# EPICS alarm handler configuration: apps/caenScalerApp/alh/watchdogs_nomoller.alhConfig
GROUP    NULL                         HallC_Ops
$GUIDANCE
This alarm panel is intended to alert the operator to various problems
with controls, DAQ and other systems.  If there is some hardware or software
that you think could be included in this panel, please contact Steve Wood.
For this alarm panel to work, vmec15 must be up and healthy.  If most
everything is in an invalid or error state, then reboot vmec15.
$END
GROUP    HallC_Ops                    DataMovement
CHANNEL  DataMovement                 HCDOG_diskwatch
$GUIDANCE
The diskwatch GUI that monitors free disk space is either hung or not
running.  This GUI should be running on the DAQ console.  If it is running,
click the Quit button.  To restart the GUI, type the command "diskwatch"
into an xterm window on the DAQ console.  (Should be logged on as "cdaq").
$END
CHANNEL  DataMovement                 HCDOG_happyreaper
$GUIDANCE
The scripts that copy runs from the data disks to the Silo do not appear
to be running.  Steve Wood should be notified.  However, if there more
than, say, five green partitions in diskwatch, the situation is not
urgent, so don't wake him up in the middle of the night.
$END
GROUP    HallC_Ops                    Monitoring
CHANNEL  Monitoring                   HCDOG_ChannelArchiver
$GUIDANCE
The EPICS Channel Archiver that maintains a continuous log of controls
information is not running.  To restart, logon to jeffylab as "cvxwrks"
 and type the following commands:
	cd ~/Archives
	./stop_archiver
	./start_archiver
$END
CHANNEL  Monitoring                   HCDOG_BetaBrite
$GUIDANCE
The LED display that shows beam current and PSS status is not working
properly.  To restart, logon to jeffylab as "cvxwrks".  Do
"ps -aux | grep bcm_pss" and kill any copies of the script that are
running.  Then type "cd ~/BETABRITE/bcm ; ./bcm_pss.pl&".
$END
GROUP    HallC_Ops                    Crates
$GUIDANCE
The status of many of the counting house NIM bins and Camac crates is
monitored by passing a pulser signal through a module in each crate.
The pulser coming from each crate is connect to an input register.  If
the pulser signal stops for a given crate, an alarm will be raised,
indicating a possible power problem with the crate.
$END
CHANNEL  Crates                       HCDOG_bit0
$GUIDANCE
The watchdog signal from the top NIM bit in rack CH03B05 is not present.
This is most likely a problem with the NIM crate (loss of power or bad
modules) and should be addressed immediately.
It could also be that the master watchdog pulser has failed.  If this is the
case, then alarms should be present for other NIM bins.
$END
CHANNEL  Crates                       HCDOG_bit1
$GUIDANCE
The watchdog signal from the third NIM bin in rack CH03B05 is not present.
This is most likely a problem with the NIM crate (loss of power or bad
modules) and should be addressed immediately.
It could also be that the master watchdog pulser has failed.  If this is the
case, then alarms should be present for other NIM bins.
$END
CHANNEL  Crates                       HCDOG_bit2
$GUIDANCE
The watchdog signal from the top NIM bin (under the CAMAC crate) in rack
CH03B06 is not present.  This is most likely a problem with the NIM crate
(loss of power or bad modules) and should be addressed immediately.
It could also be that the master watchdog pulser has failed.  If this is the
case, then alarms should be present for other NIM bins.
$END
CHANNEL  Crates                       HCDOG_bit3
$GUIDANCE
The watchdog signal from the top NIM bin CH03B07 is not present.  This
is most likely a problem with the NIM crate (loss of power or bad
modules) and should be addressed immediately.  It could also be that
the master watchdog pulser has failed.  If this is the case, then
alarms should be present for other NIM bins.
$END
INCLUDE HallC_Ops moller.alhConfig
